// SIMATIC S7-200 project (STEP 7-Micro/WIN), CPU 224XP REL 02.01

SYMBOL_TABLE USER1
s1               I0.0
s2               I0.1
reset            I0.3
do               Q0.0
xanh             Q0.1
END_SYMBOL_TABLE

ORGANIZATION_BLOCK MAIN:OB1
TITLE=PROGRAM COMMENTS
BEGIN
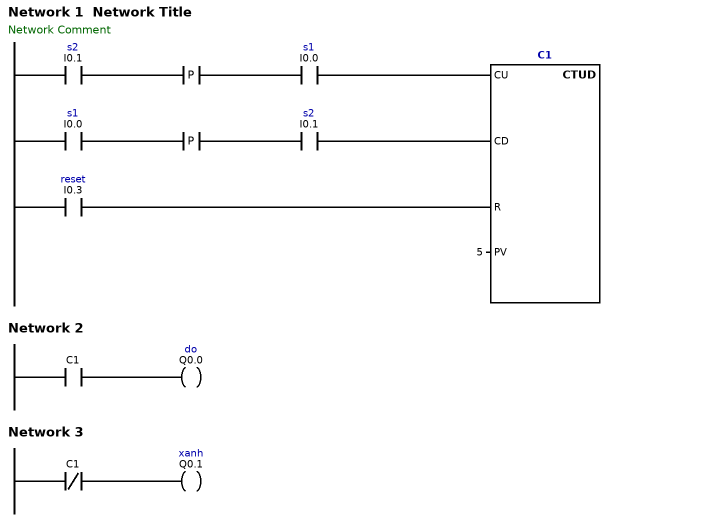
Network 1 // Network Title
// Network Comment
LD     s2:I0.1
EU
A      s1:I0.0
LD     s1:I0.0
EU
A      s2:I0.1
LD     reset:I0.3
CTUD   C1, 5
Network 2
LD     C1
=      do:Q0.0
Network 3
LDN    C1
=      xanh:Q0.1
END_ORGANIZATION_BLOCK
